(*
Nazwa:			FB_CycleTimes
Opis:			czasy cyklów
Wersja:			v0.1
Data:			2019-08-29
Autor:			DP
Urzadzenia:		
Konfiguracja:	
Info: 
- dodano opcje przesuwu liniowego
*)
FUNCTION_BLOCK FB_CycleTimes
VAR_INPUT
	bEnable: BOOL;				//Zezwolenie na pracę
	bReset:BOOL;				//Stop awaryjny nieaktywny
	tStation1CT:TIME;			//Czas cyklu stacji nr 1
	bStation1En:BOOL;			//Zezwolenie pracy stacji nr 1
	sStation1Name:STRING;		//Nazwa stacji nr 1
	tStation2CT:TIME;			//Czas cyklu stacji nr 2
	bStation2En:BOOL;			//Zezwolenie pracy stacji nr 2
	sStation2Name:STRING;		//Nazwa stacji nr 2
	tStation3CT:TIME;			//Czas cyklu stacji nr 3
	bStation3En:BOOL;			//Zezwolenie pracy stacji nr 3
	sStation3Name:STRING;		//Nazwa stacji nr 3
	tStation4CT:TIME;			//Czas cyklu stacji nr 4
	bStation4En:BOOL;			//Zezwolenie pracy stacji nr 4
	sStation4Name:STRING;		//Nazwa stacji nr 4
	tStation5CT:TIME;			//Czas cyklu stacji nr 5
	bStation5En:BOOL;			//Zezwolenie pracy stacji nr 5
	sStation5Name:STRING;		//Nazwa stacji nr 5
	tStation6CT:TIME;			//Czas cyklu stacji nr 6
	bStation6En:BOOL;			//Zezwolenie pracy stacji nr 6
	sStation6Name:STRING;		//Nazwa stacji nr 6
	tStation7CT:TIME;			//Czas cyklu stacji nr 7
	bStation7En:BOOL;			//Zezwolenie pracy stacji nr 7
	sStation7Name:STRING;		//Nazwa stacji nr 7
	tStation8CT:TIME;			//Czas cyklu stacji nr 8
	bStation8En:BOOL;			//Zezwolenie pracy stacji nr 8
	sStation8Name:STRING;		//Nazwa stacji nr 8
	tStation9CT:TIME;			//Czas cyklu stacji nr 9
	bStation9En:BOOL;			//Zezwolenie pracy stacji nr 9
	sStation9Name:STRING;		//Nazwa stacji nr 9
	tStation10CT:TIME;			//Czas cyklu stacji nr 10
	bStation10En:BOOL;			//Zezwolenie pracy stacji nr 10
	sStation10Name:STRING;		//Nazwa stacji nr 10
	tStation11CT:TIME;			//Czas cyklu stacji nr 11
	bStation11En:BOOL;			//Zezwolenie pracy stacji nr 11
	sStation11Name:STRING;		//Nazwa stacji nr 11
	tStation12CT:TIME;			//Czas cyklu stacji nr 12
	bStation12En:BOOL;			//Zezwolenie pracy stacji nr 12
	sStation12Name:STRING;		//Nazwa stacji nr 12
	tStation13CT:TIME;			//Czas cyklu stacji nr 13
	bStation13En:BOOL;			//Zezwolenie pracy stacji nr 13
	sStation13Name:STRING;		//Nazwa stacji nr 13
	tStation14CT:TIME;			//Czas cyklu stacji nr 14
	bStation14En:BOOL;			//Zezwolenie pracy stacji nr 14
	sStation14Name:STRING;		//Nazwa stacji nr 14
	tStation15CT:TIME;			//Czas cyklu stacji nr 15
	bStation15En:BOOL;			//Zezwolenie pracy stacji nr 15	
	sStation15Name:STRING;		//Nazwa stacji nr 15
	tStation16CT:TIME;			//Czas cyklu stacji nr 16
	bStation16En:BOOL;			//Zezwolenie pracy stacji nr 16	
	sStation16Name:STRING;		//Nazwa stacji nr 16
	tStation17CT:TIME;			//Czas cyklu stacji nr 17
	bStation17En:BOOL;			//Zezwolenie pracy stacji nr 17	
	sStation17Name:STRING;		//Nazwa stacji nr 17
	tStation18CT:TIME;			//Czas cyklu stacji nr 18
	bStation18En:BOOL;			//Zezwolenie pracy stacji nr 18	
	sStation18Name:STRING;		//Nazwa stacji nr 18
	tStation19CT:TIME;			//Czas cyklu stacji nr 19
	bStation19En:BOOL;			//Zezwolenie pracy stacji nr 19	
	sStation19Name:STRING;		//Nazwa stacji nr 19
	tStation20CT:TIME;			//Czas cyklu stacji nr 20
	bStation20En:BOOL;			//Zezwolenie pracy stacji nr 20	
	sStation20Name:STRING;		//Nazwa stacji nr 20



	
	
END_VAR
VAR_OUTPUT
	sSlowestStation1:STRING;		//Opis najwolniejszej stacji nr 1
	sSlowestStation2:STRING;		//Opis najwolniejszej stacji nr 2
	sSlowestStation3:STRING;		//Opis najwolniejszej stacji nr 3
	sSlowestStation4:STRING;		//Opis najwolniejszej stacji nr 4
	sSlowestStation5:STRING;		//Opis najwolniejszej stacji nr 5
	iSlowestStationCount1:INT;		//Ilość dla najwolniejszej stacji nr 1	
	iSlowestStationCount2:INT;		//Ilość dla najwolniejszej stacji nr 2		
	iSlowestStationCount3:INT;		//Ilość dla najwolniejszej stacji nr 3	
	iSlowestStationCount4:INT;		//Ilość dla najwolniejszej stacji nr 4		
	iSlowestStationCount5:INT;		//Ilość dla najwolniejszej stacji nr 5		
END_VAR

VAR
	arCycleTimes: ARRAY [1..20] OF S_CycleTimes;
	dTimeTempSlowest1:DINT;
	dTimeTempSlowest2:DINT;
	dTimeTempSlowest3:DINT;
	dTimeTempSlowest4:DINT;
	dTimeTempSlowest5:DINT;
	i: INT;
END_VAR

ErrorHandling();
Cycle();
ManualMovements();
Statistics();

ACTION Cycle:
dTimeTempSlowest1:=0;
dTimeTempSlowest2:=0;
dTimeTempSlowest3:=0;
dTimeTempSlowest4:=0;
dTimeTempSlowest5:=0;


arCycleTimes[1].bEnable:=bStation1En;
arCycleTimes[1].bName:=sStation1Name;
arCycleTimes[1].dTime:=TIME_TO_DINT(tStation1CT);
arCycleTimes[2].bEnable:=bStation2En;
arCycleTimes[2].bName:=sStation2Name;
arCycleTimes[2].dTime:=TIME_TO_DINT(tStation2CT);
arCycleTimes[3].bEnable:=bStation3En;
arCycleTimes[3].bName:=sStation3Name;
arCycleTimes[3].dTime:=TIME_TO_DINT(tStation3CT);
arCycleTimes[4].bEnable:=bStation4En;
arCycleTimes[4].bName:=sStation4Name;
arCycleTimes[4].dTime:=TIME_TO_DINT(tStation4CT);
arCycleTimes[5].bEnable:=bStation5En;
arCycleTimes[5].bName:=sStation5Name;
arCycleTimes[5].dTime:=TIME_TO_DINT(tStation5CT);
arCycleTimes[6].bEnable:=bStation6En;
arCycleTimes[6].bName:=sStation6Name;
arCycleTimes[6].dTime:=TIME_TO_DINT(tStation6CT);
arCycleTimes[7].bEnable:=bStation7En;
arCycleTimes[7].bName:=sStation7Name;
arCycleTimes[7].dTime:=TIME_TO_DINT(tStation7CT);
arCycleTimes[8].bEnable:=bStation8En;
arCycleTimes[8].bName:=sStation8Name;
arCycleTimes[8].dTime:=TIME_TO_DINT(tStation8CT);
arCycleTimes[9].bEnable:=bStation9En;
arCycleTimes[9].bName:=sStation9Name;
arCycleTimes[9].dTime:=TIME_TO_DINT(tStation9CT);
arCycleTimes[10].bEnable:=bStation10En;
arCycleTimes[10].bName:=sStation10Name;
arCycleTimes[10].dTime:=TIME_TO_DINT(tStation10CT);
arCycleTimes[11].bEnable:=bStation11En;
arCycleTimes[11].bName:=sStation11Name;
arCycleTimes[11].dTime:=TIME_TO_DINT(tStation11CT);
arCycleTimes[12].bEnable:=bStation12En;
arCycleTimes[12].bName:=sStation12Name;
arCycleTimes[12].dTime:=TIME_TO_DINT(tStation12CT);
arCycleTimes[13].bEnable:=bStation13En;
arCycleTimes[13].bName:=sStation13Name;
arCycleTimes[13].dTime:=TIME_TO_DINT(tStation13CT);
arCycleTimes[14].bEnable:=bStation14En;
arCycleTimes[14].bName:=sStation14Name;
arCycleTimes[14].dTime:=TIME_TO_DINT(tStation14CT);
arCycleTimes[15].bEnable:=bStation15En;
arCycleTimes[15].bName:=sStation15Name;
arCycleTimes[15].dTime:=TIME_TO_DINT(tStation15CT);
arCycleTimes[16].bEnable:=bStation16En;
arCycleTimes[16].bName:=sStation16Name;
arCycleTimes[16].dTime:=TIME_TO_DINT(tStation16CT);
arCycleTimes[17].bEnable:=bStation17En;
arCycleTimes[17].bName:=sStation17Name;
arCycleTimes[17].dTime:=TIME_TO_DINT(tStation17CT);
arCycleTimes[18].bEnable:=bStation18En;
arCycleTimes[18].bName:=sStation18Name;
arCycleTimes[18].dTime:=TIME_TO_DINT(tStation18CT);
arCycleTimes[19].bEnable:=bStation19En;
arCycleTimes[19].bName:=sStation19Name;
arCycleTimes[19].dTime:=TIME_TO_DINT(tStation19CT);
arCycleTimes[20].bEnable:=bStation20En;
arCycleTimes[20].bName:=sStation20Name;
arCycleTimes[20].dTime:=TIME_TO_DINT(tStation20CT);
//Dodaje na testy


FOR i:=1 TO 20 DO
	IF arCycleTimes[i].bEnable AND arCycleTimes[i].dTime > dTimeTempSlowest1 THEN
		dTimeTempSlowest1:=arCycleTimes[i].dTime;
		//sSlowestStation1:=CONCAT(arCycleTimes[i].bName,CONCAT(':',DINT_TO_STRING(dTimeTempSlowest1))); 
		sSlowestStation1:=arCycleTimes[i].bName;
		iSlowestStationCount1:=DINT_TO_INT(dTimeTempSlowest1);
	END_IF
END_FOR

FOR i:=1 TO 20 DO
	IF arCycleTimes[i].bEnable AND NOT (dTimeTempSlowest1=arCycleTimes[i].dTime) AND arCycleTimes[i].dTime > dTimeTempSlowest2 THEN
		dTimeTempSlowest2:=arCycleTimes[i].dTime;
		//sSlowestStation2:=CONCAT(arCycleTimes[i].bName,CONCAT(':',DINT_TO_STRING(dTimeTempSlowest2))); 
		sSlowestStation2:=arCycleTimes[i].bName;
		iSlowestStationCount2:=DINT_TO_INT(dTimeTempSlowest2);
	END_IF
END_FOR
	

FOR i:=1 TO 20 DO
	IF arCycleTimes[i].bEnable AND NOT (dTimeTempSlowest1=arCycleTimes[i].dTime) AND NOT (dTimeTempSlowest2=arCycleTimes[i].dTime) AND arCycleTimes[i].dTime > dTimeTempSlowest3 THEN
		dTimeTempSlowest3:=arCycleTimes[i].dTime;
		//sSlowestStation3:=CONCAT(arCycleTimes[i].bName,CONCAT(':',DINT_TO_STRING(dTimeTempSlowest3))); 
		sSlowestStation3:=arCycleTimes[i].bName;
		iSlowestStationCount3:=DINT_TO_INT(dTimeTempSlowest3);
	END_IF
END_FOR

FOR i:=1 TO 20 DO
	IF arCycleTimes[i].bEnable AND NOT (dTimeTempSlowest1=arCycleTimes[i].dTime) AND NOT (dTimeTempSlowest2=arCycleTimes[i].dTime) AND NOT (dTimeTempSlowest3=arCycleTimes[i].dTime) AND arCycleTimes[i].dTime > dTimeTempSlowest4 THEN
		dTimeTempSlowest4:=arCycleTimes[i].dTime;
		//sSlowestStation4:=CONCAT(arCycleTimes[i].bName,CONCAT(':',DINT_TO_STRING(dTimeTempSlowest4))); 
		sSlowestStation4:=arCycleTimes[i].bName;
		iSlowestStationCount4:=DINT_TO_INT(dTimeTempSlowest4);
	END_IF
END_FOR

FOR i:=1 TO 20 DO
	IF arCycleTimes[i].bEnable AND NOT (dTimeTempSlowest1=arCycleTimes[i].dTime) AND NOT (dTimeTempSlowest2=arCycleTimes[i].dTime) AND NOT (dTimeTempSlowest3=arCycleTimes[i].dTime) AND NOT (dTimeTempSlowest4=arCycleTimes[i].dTime) AND arCycleTimes[i].dTime > dTimeTempSlowest5 THEN
		dTimeTempSlowest5:=arCycleTimes[i].dTime;
		//sSlowestStation5:=CONCAT(arCycleTimes[i].bName,CONCAT(':',DINT_TO_STRING(dTimeTempSlowest5))); 
		sSlowestStation5:=arCycleTimes[i].bName;
		iSlowestStationCount5:=DINT_TO_INT(dTimeTempSlowest5);
	END_IF
END_FOR
END_ACTION

ACTION ErrorHandling:

END_ACTION

ACTION ManualMovements:

END_ACTION

ACTION Statistics:

END_ACTION

END_FUNCTION_BLOCK

(* stored: Version 1.1.0.1, ProductVersion 3.1.4026.13, FileIdentifier 6fd738f6b38d74397058905272a79bd7aaacd2fb, FileSignature a3fe1aa0adc22de2ed8205990a7ccf80b38e2e70834d7bb55001624c23c11870346d4bc44b7a43ca8071f58b0a3facd78f0cc7d5d9ed7a90fb06671fb0243fd7ab31dbe536ecfc43b55fb898e2af0ba2d9e417a0848e558f5ab1745b51af5fb9e9eb6471d423512671b0327ce23a9c726f45f71913619e1bf51c0db258af594b94130a57e02c357a92f8f2d931c3bf6194c0efc827ed8469d858ca21ea3954dccd9ba14168a77639fa27f58076509069a0b0bd4a4d8d55d8518e22a76981d8e39e3cd45739c79b99e5dd9edbbb9e04b6b169bcb79533fe5cb8b564f43f8c7f35cf393c40409215cbcc7b207a93b0e81abadaabe6c59b6388654e4fb88e613027
   POU FB_CycleTimes: Id {67d90193-0ce8-486f-9037-300071db73c9}, SpecialFunc None
   Action Cycle: Id {17f91080-9834-4ad4-8080-642fd25ddf99}
   Action ErrorHandling: Id {a9caaf0e-232b-4715-b4af-79d410dec3aa}
   Action ManualMovements: Id {03812df5-c016-4c9e-88e7-e3272e17d84c}
   Action Statistics: Id {0f7be914-8e99-4d78-bd16-4a085603642d} *)
